{attribute 'qualified_only'}
VAR_GLOBAL CONSTANT
	cNrOfAxes:					INT := 2;
	
END_VAR

VAR_GLOBAL
	stAxisRef:					ARRAY[1..cNrOfAxes] OF AXIS_REF;
	
END_VAR

(* stored: Version 1.1.0.1, ProductVersion 3.1.4024.4
   GVL GVL_IO: Id {9c4f4da1-97b5-4005-aee4-d96ad60075fe} *)
